PROGRAM MAIN
VAR
	bStartCounter : BOOL;
	nCounter : INT;
	fResult : REAL;
END_VAR


IF bStartCounter THEN
	nCounter := nCounter + 1;
ELSE
	nCounter := 0;
END_IF

END_PROGRAM

(* stored: Version 1.1.0.1, ProductVersion 3.1.4024.9
   POU MAIN: Id {02d379f3-f69d-4b07-82ff-0d9c24519264}, SpecialFunc None *)
